// TIA Portal V17 export
// export: Created 2026-07-06T15:33:03.4099563Z, ExportSetting WithDefaults, DisplayName Totally Integrated Automation Portal, DisplayVersion V17, DisplayName TIA Portal Openness, DisplayVersion V17, DisplayName TIA Portal Version Control Interface, DisplayVersion V17, DisplayName STEP 7 Professional, DisplayVersion V17, DisplayName STEP 7 Safety, DisplayVersion V17, DisplayName WinCC Professional, DisplayVersion V17
DATA_BLOCK "kinco_tcon_DB"   // DB7
// stored: AutoNumber true, DBAccessibleFromOPCUA true, InstanceOfName TCON, OfSystemLibElement TCON, OfSystemLibVersion 4.0
"TCON"
   // VAR_INPUT
   //    REQ : Bool;
   //    ID : CONN_OUC;
   // END_VAR
   // VAR_OUTPUT
   //    DONE : Bool;
   //    BUSY : Bool;
   //    ERROR : Bool;
   //    STATUS : Word;
   // END_VAR
   // VAR_IN_OUT
   //    CONNECT : Variant;
   // END_VAR
BEGIN
END_DATA_BLOCK
